/// Implicitly generated code : DO NOT EDIT
/// Checks for division by 0, if divisor is 0, replace it with 1 and report error
{attribute 'check_div_real32' := ''}
{attribute 'no_check' := ''}
FUNCTION CheckDivReal : REAL
VAR_INPUT
	divisor: REAL;
END_VAR

IF divisor = 0 THEN
	// replace divisor and report error if necessary
	CheckDivReal := 1;
	Services.fbEventHandler.Select(TC_Events.CodeEventClass.ErrorEvent)
						   .ArgSetString('div 0 REAL')
						   .Raise();
ELSE
	CheckDivReal := divisor;
END_IF;

END_FUNCTION

(* stored: Version 1.1.0.1
   POU CheckDivReal: Id {f9e6042d-68ce-4364-8be8-09f8d3ecf106}, SpecialFunc None *)
